VAR_GLOBAL
	sTextBox : STRING;
	sInput : STRING;
	sPWInput : STRING;
	rNumericInput : REAL;
END_VAR

(* stored: Version 1.1.0.1, ProductVersion 3.1.4024.12
   GVL GVL: Id {ea6f89fe-c956-4ab1-813b-0ffb0e4fafcd} *)
